(* Logix 5000 project; controller TRN_ICP_RA5000_AIO 1769-L16ER-BB1B rev 33.11; software revision 33.00 *)

TASK MainTask (continuous, watchdog 500 ms) : MainProgram

MODULES
   Local : 1769-L16ER-BB1B (PointIO 0, rev 33.11)
      Discrete_IO : Embedded (PointIO 1, rev 33.11, Output RPI 20 ms)
           Local:1:O.Data.0   // Green light
           Local:1:O.Data.1   // Yellow light
           Local:1:O.Data.2   // Red Light
           Local:1:O.Data.3   // Blue light
           Local:1:I.Data.0   // Green Button
           Local:1:I.Data.1   // Yellow button
           Local:1:I.Data.2   // Red button
           Local:1:I.Data.4   // Switch 1
           Local:1:I.Data.3   // Blue button
END_MODULES

VAR_GLOBAL   (* controller tags *)
   LightTimer : TIMER := (PRE := 4000, ACC := 3190, EN := 1, TT := 1);
END_VAR

PROGRAM MainProgram   (* main routine MainRoutine *)

ROUTINE MainRoutine   (* ladder *)
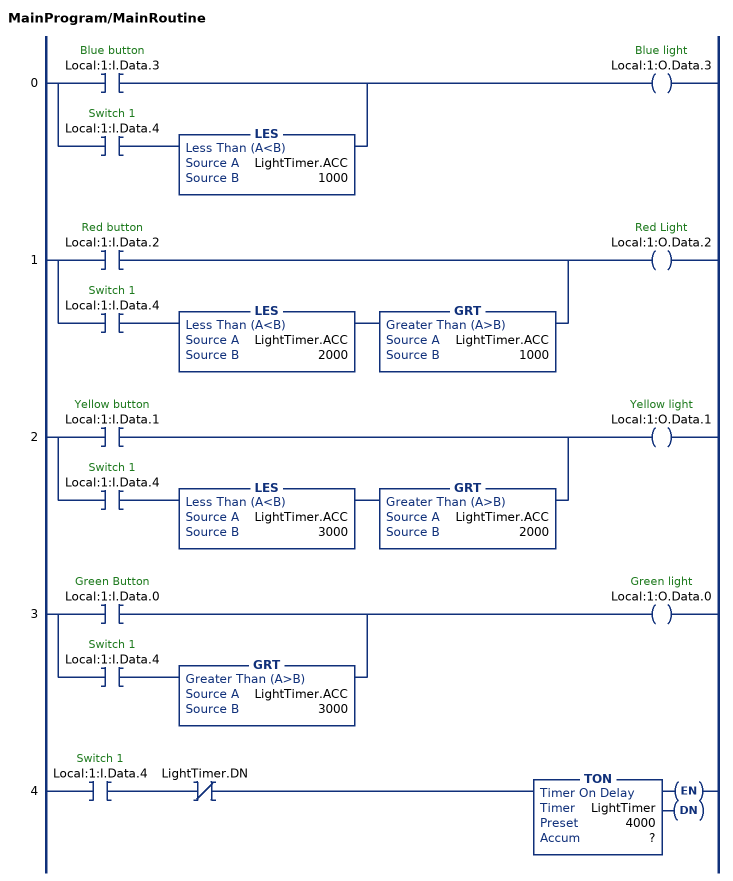
   0: [XIC(Local:1:I.Data.3) ,XIC(Local:1:I.Data.4) LES(LightTimer.ACC,1000) ]OTE(Local:1:O.Data.3);
   1: [XIC(Local:1:I.Data.2) ,XIC(Local:1:I.Data.4) LES(LightTimer.ACC,2000) GRT(LightTimer.ACC,1000) ]OTE(Local:1:O.Data.2);
   2: [XIC(Local:1:I.Data.1) ,XIC(Local:1:I.Data.4) LES(LightTimer.ACC,3000) GRT(LightTimer.ACC,2000) ]OTE(Local:1:O.Data.1);
   3: [XIC(Local:1:I.Data.0) ,XIC(Local:1:I.Data.4) GRT(LightTimer.ACC,3000) ]OTE(Local:1:O.Data.0);
   4: XIC(Local:1:I.Data.4)XIO(LightTimer.DN)TON(LightTimer,?,?);
END_ROUTINE
END_PROGRAM
